TYPE HandlingComSubscribe :
STRUCT
  Request : HandlingComRequest; // contains booleans that are used to start a specific sequence.
  Equipment : HandlingComSubscribeEquipment;  // structs for equipment objects which are used by the bridges
END_STRUCT
END_TYPE

(* stored: Version 1.1.0.1
   DUT HandlingComSubscribe: Id {af71f8c2-b674-4d62-a018-4ffb9293a4aa} *)
